Staubli VAL3: Save.pgx

program Save()
  local num l_ni
begin
  //
  libSave()
  popUpMsg("保存完毕!")
end
